FUNCTION_BLOCK FB_LocalSystemTimeProvider IMPLEMENTS I_LocalSystemTimeProvider
VAR
	_localSystemTime			: Tc2_Utilities.FB_LocalSystemTime;
	_currentSystemTimeInfo		: ST_CurrentSystemTimeInfo;
	_dateTimeToStringCovnerter	: FB_DateTimeToStringConverter;
	_iDateTimeToStringConverter	: I_DateTimeToStringConverter := _dateTimeToStringCovnerter;
END_VAR

_localSystemTime(
	sNetID:= '', 
	bEnable:= TRUE, 
	dwCycle:= 1, 
	systemTime=> _currentSystemTimeInfo.Value);
	
_currentSystemTimeInfo.IsValid := _currentSystemTimeInfo.Value.wYear > 1970;
	
_dateTimeToStringCovnerter(
	localSystemTime := _localSystemTime);

METHOD PUBLIC ConvertToString : I_DateTimeToStringConverter
VAR_INPUT
END_VAR
ConvertToString := _iDateTimeToStringConverter;
END_METHOD

{attribute 'monitoring':='call'}
// Gets current system timo info as a <ST_CurrentSystemTimeInfo>
PROPERTY CurrentTime : REFERENCE TO ST_CurrentSystemTimeInfo
GET
CurrentTime REF= _currentSystemTimeInfo;
END_GET
END_PROPERTY

// Sets the system time. Returns TRUE when done.
METHOD SetSystemTime : BOOL
VAR_INPUT
	timeToSet	: Tc2_Utilities.TIMESTRUCT;
END_VAR

VAR_OUTPUT
	error	: BOOL;	// Will be TRUE if an error occurs
	errorId	: TcError.AdsErrorCodes;	// Error code is reported here
END_VAR

VAR_INST
	setLocalTime	: Tc2_Utilities.NT_SetLocalTime :=(
		NETID := '',
		TMOUT := Tc2_System.DEFAULT_ADS_TIMEOUT);
	requestActive	: BOOL;
END_VAR
IF NOT requestActive THEN
	requestActive := TRUE;
	setLocalTime(START := FALSE);
ELSE
	setLocalTime(START := TRUE, NETID := '', TIMESTR := timeToSet);
	IF setLocalTime.BUSY = FALSE THEN
		setLocalTime(START := FALSE);
		requestActive := FALSE;
		SetSystemTime := TRUE;
	END_IF
END_IF

errorId := TcError.ToAdsErrorCode(TcError.ToAdsErrorCode(setLocalTime.ERRID));
error := setLocalTime.ERR;
END_METHOD

END_FUNCTION_BLOCK

(* stored: Version 1.1.0.1, ProductVersion 3.1.4024.15
   POU FB_LocalSystemTimeProvider: Id {5429ddc3-78d0-058e-1e56-29d8805b55eb}, SpecialFunc None
   Method ConvertToString: Id {58bacec0-cbb6-06a5-2496-f57f6a7d0a7f}
   Property CurrentTime: Id {6c4e9ddf-27e1-0836-04f5-9138aa3c0289}
   Get Get: Id {1dc69109-a2fc-07e6-33f1-0d17b5b22722}
   Method SetSystemTime: Id {2f058135-c7bf-0153-2332-c6df018c6368} *)
